FUNCTION F_AND_REF_EX : BOOL
VAR_IN_OUT
	bValueRoot		: BOOL;	
END_VAR
VAR_INPUT
	bValueCombine	: BOOL;
	bInitialize		: BOOL;
END_VAR

IF bInitialize THEN
	bValueRoot := TRUE;
END_IF
	
F_AND_REF(bValueRoot, bValueCombine);

END_FUNCTION

(* stored: Version 1.1.0.1, ProductVersion 3.1.4024.11
   POU F_AND_REF_EX: Id {211554ca-9131-4554-a35a-598dbfb8a439}, SpecialFunc None *)
